{attribute 'GeneratedUsingTerminal: EL2212-0000-0018'}
{attribute addProperty BoxType "EL2212-0000-0018"}
{attribute addProperty Id "DOX_Status_Channel_1AT %I*DOX_Status_Channel_09DD45C87DOX_Status_Channel_2AT %I*DOX_Status_Channel_09DD45C87DOX_Control_Channel_1AT %Q*DOX_Control_Channel_A74F23633DOX_Control_Channel_2AT %Q*DOX_Control_Channel_A74F23633WcStateAT %I*WcState_9091E0EB2InfoDataAT %I*InfoData_94A18F5E2"}
{attribute addProperty CRC "1171379232"}
{attribute addProperty Size "24"}
TYPE EL2212_45D1D420 EXTENDS EtcSlaveTerminalBase_947E5A46 :
STRUCT
	{attribute addProperty Name "DOX_Status_Channel_1"}
	DOX_Status_Channel_1 : DOX_Status_Channel_09DD45C8;
	{attribute addProperty Name "DOX_Status_Channel_2"}
	DOX_Status_Channel_2 : DOX_Status_Channel_09DD45C8;
	{attribute addProperty Name "DOX_Control_Channel_1"}
	DOX_Control_Channel_1 : DOX_Control_Channel_A74F2363;
	{attribute addProperty Name "DOX_Control_Channel_2"}
	DOX_Control_Channel_2 : DOX_Control_Channel_A74F2363;
	{attribute addProperty Name "WcState"}
	WcState : WcState_9091E0EB;
	{attribute addProperty Name "InfoData"}
	InfoData : InfoData_94A18F5E;
END_STRUCT
END_TYPE

(* stored: Version 1.2.0.0, ProductVersion 3.1.4024.9
   DUT EL2212_45D1D420: Id {97406cb1-9d8d-42a1-9931-8f52955b50e8} *)
